FUNCTION_BLOCK TESTING EXTENDS FB_STATION
VAR_INPUT
END_VAR
VAR_OUTPUT
END_VAR
VAR
END_VAR

ACTION A_SFC:
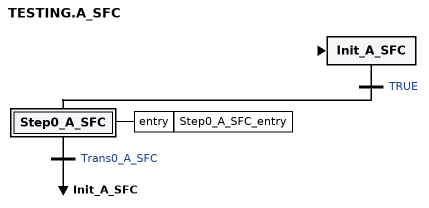
STEP Init_A_SFC:
END_STEP
TRANSITION FROM Init_A_SFC TO Step0_A_SFC
    := TRUE;
END_TRANSITION
INITIAL_STEP Step0_A_SFC:
    Step0_A_SFC_entry(P1);  // entry action
END_STEP
TRANSITION FROM Step0_A_SFC TO Init_A_SFC
    := Trans0_A_SFC;
END_TRANSITION
END_ACTION

ACTION Step0_A_SFC_entry:

END_ACTION

END_FUNCTION_BLOCK

(* stored: Version 1.1.0.1, ProductVersion 3.1.4024.12
   POU TESTING: Id {e2e2414b-9803-45f7-a0c2-b1717a8eb4d2}, SpecialFunc None
   Action A_SFC: Id {69c5a410-02f8-4e47-a778-685cd9592910}
   Action Step0_A_SFC_entry: Id {3d424d34-7c9f-4a2b-afc9-d39f221bc42a} *)
